(*
A list implementation for managing `I_Arg`.  
*)
FUNCTION_BLOCK ArgList
VAR_GENERIC CONSTANT
	nCap	: UDINT := 100;
END_VAR

IMPLEMENTS I_MutArgList

VAR
	_iList	: ARRAY[1..nCap] OF I_Arg;
END_VAR

(*
Provides the maximum capacity of the list.
*)
PROPERTY Cap : UDINT
GET
Cap := nCap;
END_GET
END_PROPERTY

(*
Retrieves the `I_Arg` at the specified index.  
Returns:
- `Ok` - Successfully retrieves the `I_Arg`.
- `Err.Idx` - The specified index is out of bounds.
*)
METHOD Get : Result
VAR_INPUT
	nIndex		: UDINT;
END_VAR
VAR_OUTPUT
	iArg	: I_Arg;
END_VAR
IF nIndex > nCap OR nIndex = 0 THEN
	Get := Err.Idx;
	RETURN;	
END_IF

iArg := _iList[nIndex];
IF iArg <> 0 THEN
	Get := Ok;
END_IF
END_METHOD

(*
Adds, updates, or removes an argument in the list at the specified index.  
Return:
- `Ok` - Upon successfully adding, modifying, or removing an entry.
- `Err.Idx` - When attempting to modify an entry at an out-of-bounds index.
*)
METHOD Set : Result
VAR_INPUT
	iArg		: I_Arg;
	nIndex		: UDINT;
END_VAR
IF nIndex > nCap OR nIndex = 0 THEN
	Set := Err.Idx;
	RETURN;	
END_IF

_iList[nIndex] := iArg;
IF iArg <> 0 THEN
	Set := Ok;
END_IF
END_METHOD

END_FUNCTION_BLOCK

(* stored: Version 1.1.0.1
   POU ArgList: Id {2b96f983-70e4-40e0-8445-dead91093f2f}, SpecialFunc None
   Property Cap: Id {1048cc8b-e43e-4da9-a171-782c39431c37}
   Get Get: Id {c0c3415d-8c77-4181-aeea-f218ef2d28f8}
   Method Get: Id {5c57983f-1819-44e3-afe2-2f589f56d44d}
   Method Set: Id {e43a485e-6cb6-45fe-b385-9a9421cc55b9} *)
